# EPICS substitutions: iocs/bcur/iocBoot/iocbcur/substitutions/canberra_3.substitutions
file "$(MCA)/mcaApp/Db/simple_mca.db"
{
pattern
{P           M       DTYP           INP              PREC  CHANS}
{bcur:med:   mca1  "asynMCA"       "@asyn(AIM1/1 0)"  3     2048}
{bcur:med:   mca2  "asynMCA"       "@asyn(AIM1/2 0)"  3     2048}
{bcur:med:   mca3  "asynMCA"       "@asyn(AIM2/1 0)"  3     2048}
{bcur:med:   mca0  "Soft Channel"  ""                 3     2048}
}

#file "$(MCA)/mcaApp/Db/icb_amp.db"
#{
#pattern
#{P			AMP		PORT}
#{bcur:med:	amp1	icbAmp1}
#}

file "$(MCA)/mcaApp/Db/icb_adc.db"
{
pattern
{P			ADC		PORT}
{bcur:med:	adc1	"icbAdc1"}
{bcur:med:	adc2	"icbAdc2"}
{bcur:med:	adc3	"icbAdc3"}
}

#file "$(MCA)/mcaApp/Db/icb_hvps.db"
#{
#pattern
#{P			HVPS	LIMIT	PORT}
#{bcur:med:	hvps1	1000	"icbHvps1"}
#}

file "$(MCA)/mcaApp/Db/icb_tca.db"
{
pattern
{P,          TCA,	PORT,		MCA}
{bcur:med:,  tca1,	"icbTca1",	mca1}
{bcur:med:,  tca2,	"icbTca2",	mca2}
{bcur:med:,  tca3,	"icbTca3",	mca3}
}
